// TIA Portal V21 export
// export: Created 2026-08-23T01:33:54.3053779Z, ExportSetting WithDefaults, DisplayName Totally Integrated Automation Portal, DisplayVersion V21, DisplayName SINAMICS Startdrive Advanced, DisplayVersion V21, DisplayName SINAMICS Startdrive G110M, G120, G120C, G120D, G120P, G115D, DisplayVersion V21, DisplayName SINAMICS Startdrive G130, G150, S120, S150, G200, G220, S200, S210, S220, Innomotics MVD, DisplayVersion V21, DisplayName STEP 7 Professional, DisplayVersion V21, DisplayName STEP 7 Safety, DisplayVersion V21, DisplayName Tech WebApplication, DisplayVersion V21, DisplayName WinCC Basic/Comfort/Advanced, DisplayVersion V21, DisplayName WinCC Unified, DisplayVersion V21
FUNCTION_BLOCK "FB_GraphDemo"   // FB2, GRAPH
VERSION : 0.1
// stored: AcknowledgeErrorsRequired true, AutoNumber true, GraphVersion 6.0, InitialValuesAcquisition false, IsIECCheckEnabled false, LanguageInNetworks LAD, LockOperatingMode false, PermanentILProcessingInMANMode false, SetENOAutomatically false, SkipSteps false, UDAEnableTagReadback false, WithAlarmHandling true
   // inherited from GRAPH_BASE
   VAR
      OFF_SQ_BASE : Bool;
   END_VAR
   VAR_INPUT
      OFF_SQ : Bool := false;   // Turn sequence off
      INIT_SQ : Bool := false;   // Set sequence to initial state
      ACK_EF : Bool := false;   // Acknowledge all errors and faults
      Cond1 : Bool;
      Cond2 : Bool;
   END_VAR
   VAR_OUTPUT
      Out1 : Bool;
      Out2 : Bool;
      Out3 : Bool;
   END_VAR
BEGIN
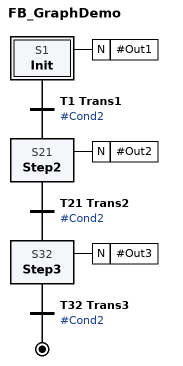
   // sequencer 1
   INITIAL_STEP Init:   // S1, max time T#10S, warning time T#7S
      interlock C := #Cond2;
      supervision V := #Cond1;
              N    #Out1
   END_STEP
   TRANSITION Trans1 FROM Init TO Step2   // T1
      := #Cond2;
   END_TRANSITION
   STEP Step2:   // S21, max time T#10S, warning time T#7S
      interlock C := #Cond2;
      supervision V := #Cond1;
              N    #Out2
   END_STEP
   TRANSITION Trans2 FROM Step2 TO Step3   // T21
      := #Cond2;
   END_TRANSITION
   STEP Step3:   // S32, max time T#10S, warning time T#7S
      interlock C := #Cond2;
      supervision V := #Cond1;
              N    #Out3
   END_STEP
   TRANSITION Trans3 FROM Step3 TO END   // T32
      := #Cond2;
   END_TRANSITION
END_FUNCTION_BLOCK
